{attribute 'qualified_only'}
{attribute 'strict'}
TYPE EWPWeight :
(
	light :=1,
	medium := 2,
	heavy := 3,
	undetermined :=4,
	enum_member := 0
);
END_TYPE

(* stored: Version 1.1.0.1, ProductVersion 3.1.4024.9
   DUT EWPWeight: Id {1b9916d8-3b42-4b35-afcc-78ae89ba3bbc} *)
